FUNCTION_BLOCK FB_Conveyor
VAR
    bConveyorRunning : BOOL;
END_VAR

GVL.g_bConveyorMotor := bConveyorRunning;

METHOD Start
 bConveyorRunning := TRUE;
END_METHOD

METHOD Stop
 bConveyorRunning := FALSE;
END_METHOD

END_FUNCTION_BLOCK

(* stored: Version 1.1.0.1, ProductVersion 3.1.4024.16
   POU FB_Conveyor: Id {5188e069-9cdf-45ef-a19f-f2cd5b6e0bd9}, SpecialFunc None
   Method Start: Id {43287206-e450-4847-af4b-2a6d2462f53d}
   Method Stop: Id {62652d42-7838-44c8-bd67-1a6cd2cbea3f} *)
